// TIA Portal V19 export
FUNCTION_BLOCK "Simulation"   // FB1, LAD
{ S7_Optimized_Access := 'TRUE' }
// stored: MemoryReserve 100, SetENOAutomatically false
   VAR
      LGF_Error : Array[1..10] of Bool;
      LGF_Status : Array[1..10] of Word;
      RetValReal : Real;
   END_VAR
   VAR_TEMP
      RndDIntStatus : Array[1..10] of Word;
      RndRealStatus : Array[1..10] of Word;
   END_VAR
   VAR_TEMP   // added for the SCL form of the ladder/FBD networks
      _w1 : Bool;
      _w2 : Bool;
      _w3 : Bool;
   END_VAR
BEGIN

REGION Network 1: Sensor simulation Machine 1
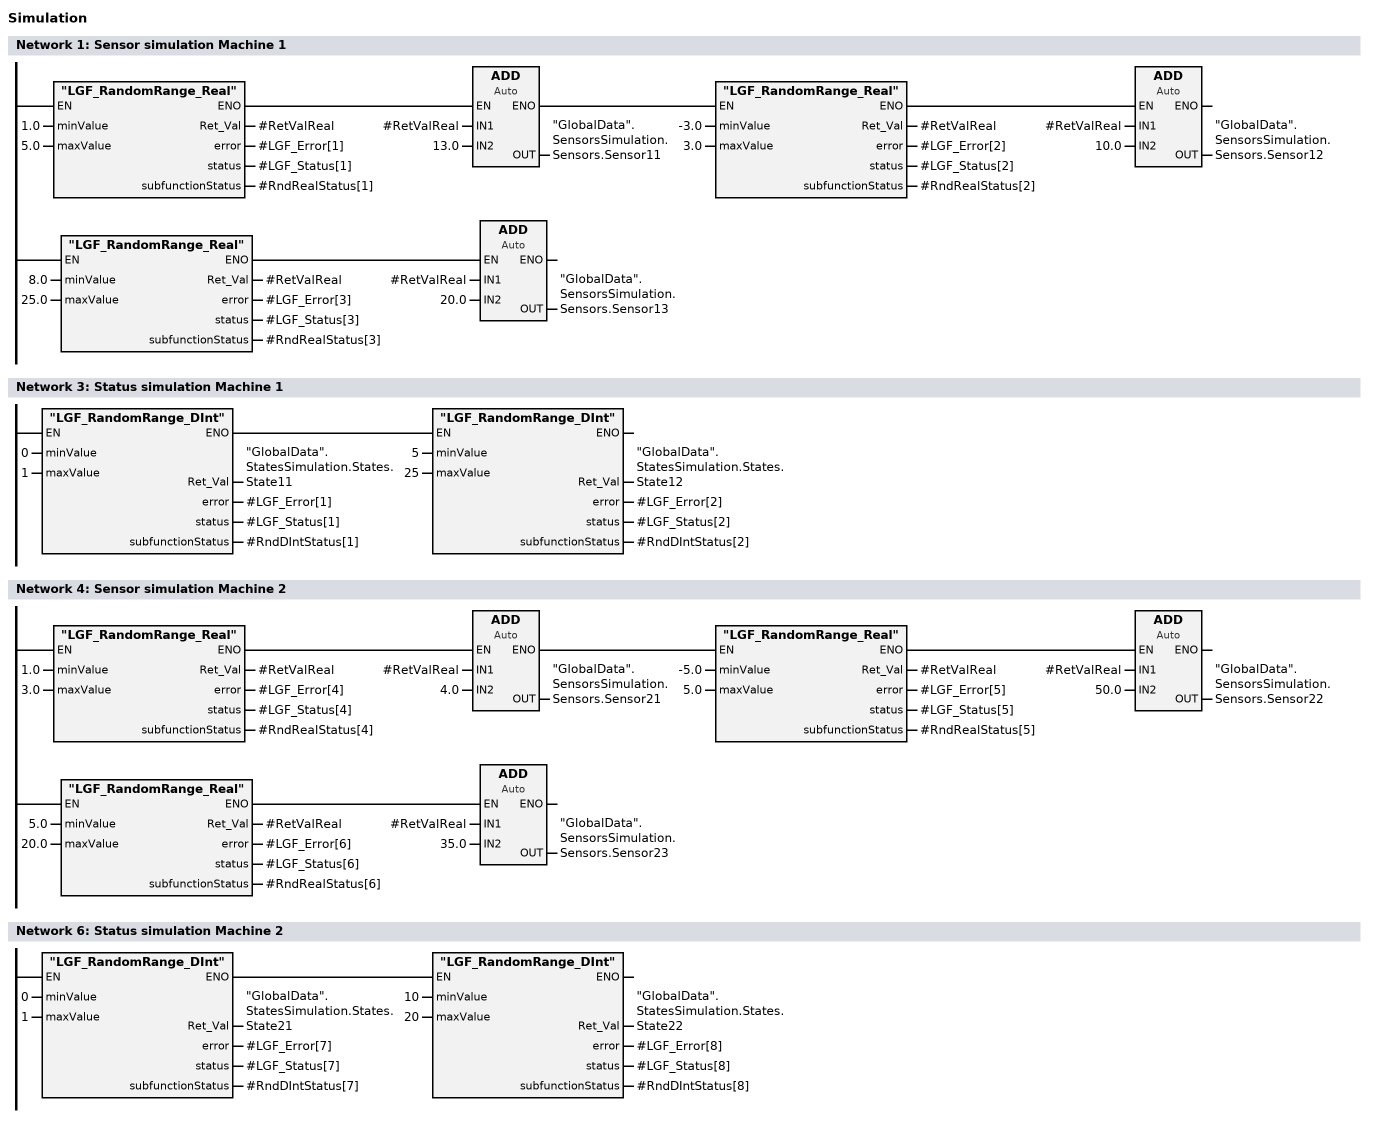
   RUNG wire#powerrail
      "LGF_RandomRange_Real"(minValue := 1.0, maxValue := 5.0, Ret_Val => #RetValReal, error => #LGF_Error[1], status => #LGF_Status[1], subfunctionStatus => #RndRealStatus[1])
      Add(in1 := #RetValReal, in2 := 13.0, out => "GlobalData".SensorsSimulation.Sensors.Sensor11)
      "LGF_RandomRange_Real"(minValue := -3.0, maxValue := 3.0, Ret_Val => #RetValReal, error => #LGF_Error[2], status => #LGF_Status[2], subfunctionStatus => #RndRealStatus[2])
      Add(in1 := #RetValReal, in2 := 10.0, out => "GlobalData".SensorsSimulation.Sensors.Sensor12)
   END_RUNG
   RUNG wire#powerrail
      "LGF_RandomRange_Real"(minValue := 8.0, maxValue := 25.0, Ret_Val => #RetValReal, error => #LGF_Error[3], status => #LGF_Status[3], subfunctionStatus => #RndRealStatus[3])
      Add(in1 := #RetValReal, in2 := 20.0, out => "GlobalData".SensorsSimulation.Sensors.Sensor13)
   END_RUNG
   // the same network as SCL:
   #RetValReal := "LGF_RandomRange_Real"(minValue := 1.0,
                           maxValue := 5.0,
                           error => #LGF_Error[1],
                           status => #LGF_Status[1],
                           subfunctionStatus => #RndRealStatus[1],
                           ENO => #_w1);
   IF #_w1 THEN "GlobalData".SensorsSimulation.Sensors.Sensor11 := #RetValReal + 13.0; END_IF;
   #RetValReal := "LGF_RandomRange_Real"(EN := #_w1,
                           minValue := -3.0,
                           maxValue := 3.0,
                           error => #LGF_Error[2],
                           status => #LGF_Status[2],
                           subfunctionStatus => #RndRealStatus[2],
                           ENO => #_w2);
   IF #_w2 THEN "GlobalData".SensorsSimulation.Sensors.Sensor12 := #RetValReal + 10.0; END_IF;
   #RetValReal := "LGF_RandomRange_Real"(minValue := 8.0,
                           maxValue := 25.0,
                           error => #LGF_Error[3],
                           status => #LGF_Status[3],
                           subfunctionStatus => #RndRealStatus[3],
                           ENO => #_w3);
   IF #_w3 THEN "GlobalData".SensorsSimulation.Sensors.Sensor13 := #RetValReal + 20.0; END_IF;
END_REGION

REGION Network 2 (SCL): Sensor simulation Machine 1
   "GlobalData".SensorsSimulation.Sensors.Sensor14 := "GlobalData".SensorsSimulation.Sensors.Sensor14 + 0.01;

   IF "GlobalData".SensorsSimulation.Sensors.Sensor14 > 100 THEN
       "GlobalData".SensorsSimulation.Sensors.Sensor14 := 0;
   END_IF;
END_REGION

REGION Network 3: Status simulation Machine 1
   RUNG wire#powerrail
      "LGF_RandomRange_DInt"(minValue := 0, maxValue := 1, Ret_Val => "GlobalData".StatesSimulation.States.State11, error => #LGF_Error[1], status => #LGF_Status[1], subfunctionStatus => #RndDIntStatus[1])
      "LGF_RandomRange_DInt"(minValue := 5, maxValue := 25, Ret_Val => "GlobalData".StatesSimulation.States.State12, error => #LGF_Error[2], status => #LGF_Status[2], subfunctionStatus => #RndDIntStatus[2])
   END_RUNG
   // the same network as SCL:
   "GlobalData".StatesSimulation.States.State11 := "LGF_RandomRange_DInt"(minValue := 0,
                           maxValue := 1,
                           error => #LGF_Error[1],
                           status => #LGF_Status[1],
                           subfunctionStatus => #RndDIntStatus[1],
                           ENO => #_w1);
   IF #_w1 THEN
       "GlobalData".StatesSimulation.States.State12 := "LGF_RandomRange_DInt"(minValue := 5,
                               maxValue := 25,
                               error => #LGF_Error[2],
                               status => #LGF_Status[2],
                               subfunctionStatus => #RndDIntStatus[2]);
   END_IF;
END_REGION

REGION Network 4: Sensor simulation Machine 2
   RUNG wire#powerrail
      "LGF_RandomRange_Real"(minValue := 1.0, maxValue := 3.0, Ret_Val => #RetValReal, error => #LGF_Error[4], status => #LGF_Status[4], subfunctionStatus => #RndRealStatus[4])
      Add(in1 := #RetValReal, in2 := 4.0, out => "GlobalData".SensorsSimulation.Sensors.Sensor21)
      "LGF_RandomRange_Real"(minValue := -5.0, maxValue := 5.0, Ret_Val => #RetValReal, error => #LGF_Error[5], status => #LGF_Status[5], subfunctionStatus => #RndRealStatus[5])
      Add(in1 := #RetValReal, in2 := 50.0, out => "GlobalData".SensorsSimulation.Sensors.Sensor22)
   END_RUNG
   RUNG wire#powerrail
      "LGF_RandomRange_Real"(minValue := 5.0, maxValue := 20.0, Ret_Val => #RetValReal, error => #LGF_Error[6], status => #LGF_Status[6], subfunctionStatus => #RndRealStatus[6])
      Add(in1 := #RetValReal, in2 := 35.0, out => "GlobalData".SensorsSimulation.Sensors.Sensor23)
   END_RUNG
   // the same network as SCL:
   #RetValReal := "LGF_RandomRange_Real"(minValue := 1.0,
                           maxValue := 3.0,
                           error => #LGF_Error[4],
                           status => #LGF_Status[4],
                           subfunctionStatus => #RndRealStatus[4],
                           ENO => #_w1);
   IF #_w1 THEN "GlobalData".SensorsSimulation.Sensors.Sensor21 := #RetValReal + 4.0; END_IF;
   #RetValReal := "LGF_RandomRange_Real"(EN := #_w1,
                           minValue := -5.0,
                           maxValue := 5.0,
                           error => #LGF_Error[5],
                           status => #LGF_Status[5],
                           subfunctionStatus => #RndRealStatus[5],
                           ENO => #_w2);
   IF #_w2 THEN "GlobalData".SensorsSimulation.Sensors.Sensor22 := #RetValReal + 50.0; END_IF;
   #RetValReal := "LGF_RandomRange_Real"(minValue := 5.0,
                           maxValue := 20.0,
                           error => #LGF_Error[6],
                           status => #LGF_Status[6],
                           subfunctionStatus => #RndRealStatus[6],
                           ENO => #_w3);
   IF #_w3 THEN "GlobalData".SensorsSimulation.Sensors.Sensor23 := #RetValReal + 35.0; END_IF;
END_REGION

REGION Network 5 (SCL): Sensor simulation Machine 2
   "GlobalData".SensorsSimulation.Sensors.Sensor24 := "GlobalData".SensorsSimulation.Sensors.Sensor24 + 0.1;

   IF "GlobalData".SensorsSimulation.Sensors.Sensor24 > 50 THEN
       "GlobalData".SensorsSimulation.Sensors.Sensor24 := 0;
   END_IF;
END_REGION

REGION Network 6: Status simulation Machine 2
   RUNG wire#powerrail
      "LGF_RandomRange_DInt"(minValue := 0, maxValue := 1, Ret_Val => "GlobalData".StatesSimulation.States.State21, error => #LGF_Error[7], status => #LGF_Status[7], subfunctionStatus => #RndDIntStatus[7])
      "LGF_RandomRange_DInt"(minValue := 10, maxValue := 20, Ret_Val => "GlobalData".StatesSimulation.States.State22, error => #LGF_Error[8], status => #LGF_Status[8], subfunctionStatus => #RndDIntStatus[8])
   END_RUNG
   // the same network as SCL:
   "GlobalData".StatesSimulation.States.State21 := "LGF_RandomRange_DInt"(minValue := 0,
                           maxValue := 1,
                           error => #LGF_Error[7],
                           status => #LGF_Status[7],
                           subfunctionStatus => #RndDIntStatus[7],
                           ENO => #_w1);
   IF #_w1 THEN
       "GlobalData".StatesSimulation.States.State22 := "LGF_RandomRange_DInt"(minValue := 10,
                               maxValue := 20,
                               error => #LGF_Error[8],
                               status => #LGF_Status[8],
                               subfunctionStatus => #RndDIntStatus[8]);
   END_IF;
END_REGION
END_FUNCTION_BLOCK
